TYPE "bwu4067CustomInput16bytes"
TITLE = {"version":"v1.0","author":"cyanezf","family":"core/controller/bihl-wiedermann/bwu4067","status":"current","deprecatedBy": null,"dependencies":["sick_ahm36_status", "sick_dx35"]}

//(*--
//# Documentation
//## Log
//| version | date | author | description |
//|:-------:|:----:|:------:|:------------|
//| v1.0 | 2025-03-03 | cyanezf | First version |
//
//## Description
//B+W - bwu4067 Custom Input 16 bytes
//--*)

   STRUCT
      p1_spare : DWord;   // Reserved Io-link port
      p2_encoder { S7_SetPoint := 'False'} : "sick_ahm36_status";   // BW4067-16bytes/Port 2-4bytes: Encoder
      p3_distance { S7_SetPoint := 'False'} : "sick_dx35";   // BW4067-16bytes/Port 3-4bytes: Distance sensor
      p4_distance { S7_SetPoint := 'False'} : "sick_dx35";   // BW4067-16bytes/Port 4-4bytes: Distance sensor
   END_STRUCT;

END_TYPE
